FUNCTION_BLOCK FB_TestDevice IMPLEMENTS I_Focus, I_Nasmyth
VAR_INPUT
END_VAR
VAR_OUTPUT
END_VAR
VAR
END_VAR

END_FUNCTION_BLOCK

(* stored: Version 1.1.0.1, ProductVersion 3.1.4024.13
   POU FB_TestDevice: Id {88d37211-e048-4fcc-a4d0-a3e1706c8869}, SpecialFunc None *)
